(* IEC 61131-3 sources: Industry-PLC-LLM/data/PLCBEAD_repo/PLCBEAD_PLCEmbed-main/PLC-BEAD/Source/GEB/DT_TO_TOD, 1 file *)

(* ---- DT_TO_TOD.ST ---- *)
FUNCTION DT_TO_TOD2:UDINT
	VAR_INPUT
		IN :	UDINT;
	END_VAR

	DT_TO_TOD2 := (IN MOD UDINT#86400) * UDINT#1000;
END_FUNCTION

PROGRAM program0
  VAR
    LocalVar0 : UDINT;
	LocalOUT  : UDINT;
  END_VAR
  	LocalOUT := DT_TO_TOD2(LocalVar0);
END_PROGRAM
